FUNCTION_BLOCK EL2008
VAR
	{attribute addProperty Name "WcState"}
	_wcState : WcStateBase;
	{attribute addProperty Name "Info data"}
	_infoData : InfoDataBase;
	_io : EL2xx8_Data;
END_VAR

PROPERTY IO : REFERENCE TO EL2xx8_Data
GET
IO REF= _io;
END_GET
END_PROPERTY

PROPERTY WcState : REFERENCE TO WcStateBase
GET
WcState REF= _wcState;
END_GET
END_PROPERTY

END_FUNCTION_BLOCK

(* stored: Version 1.1.0.1, ProductVersion 3.1.4024.9
   POU EL2008: Id {5950e863-1fda-088d-18bb-4d096c4607c1}, SpecialFunc None
   Property IO: Id {93a8bf92-fc89-0efb-0133-a62f67426657}
   Get Get: Id {b666080f-8fd3-03f6-35d3-469a4e0c19e9}
   Property WcState: Id {04e6eb73-ec5c-0c1e-03da-461c45997938}
   Get Get: Id {731629be-8866-0f19-2a0d-326c5e2aa9b6} *)
